INTERFACE ITF_ReportDataTool

METHOD Report : BOOL
VAR_INPUT
	somemessage : ARRAY[0..5] OF BYTE;
END_VAR
END_METHOD

END_INTERFACE

(* stored: Version 1.1.0.1, ProductVersion 3.1.4024.12
   Itf ITF_ReportDataTool: Id {166c5ea4-2725-476d-89d4-b639d12a711c}
   Method Report: Id {aee1e91b-ee81-46d1-9927-2ec179f4284c} *)
